Yaskawa INFORM job: A-9-08279-80-90-L.JBI

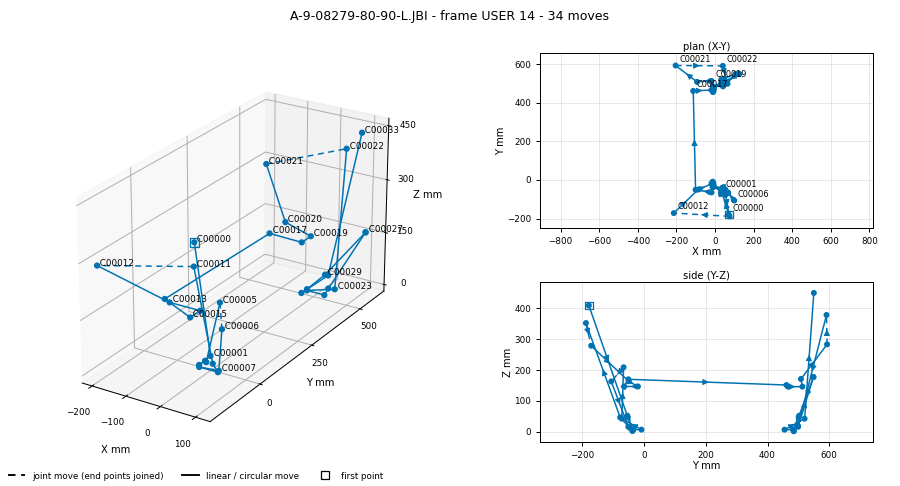
[picture p0: tool path of A-9-08279-80-90-L.JBI in frame USER 14, 34 of 34 moves have a stored position in this frame; points joined in program order, loops and branches not executed]
/JOB
//NAME A-9-08279-80-90-L
///FOLDERNAME PART_420-08279-80
//POS
///NPOS 34,0,34,0,0,0
///USER 14
///TOOL 4
///POSTYPE USER
///RECTAN
///RCONF 1,0,0,0,0,0,0,0,0,0,0,0,0,0,0,0,0,0,0,0,0,0,0,0
C00000=70.970,-178.868,409.213,-165.0000,45.0000,0.0000
C00001=33.224,-54.308,52.156,-165.0000,45.0000,0.0000
C00002=-12.412,-35.347,6.916,178.9966,57.8134,-39.3495
C00003=-12.252,-8.486,6.906,178.9975,57.8083,-39.3460
C00004=32.283,-72.150,42.455,-165.0000,45.0000,0.0000
C00005=68.685,-66.272,209.042,-165.0000,45.0000,0.0000
C00006=99.538,-106.298,163.160,-166.3780,45.3490,-50.4350
C00007=54.868,-50.966,16.241,133.5610,7.6410,-152.0390
C00008=-10.772,-37.614,2.810,126.3860,11.5189,-151.1158
C00009=43.673,-37.455,3.156,126.4274,11.4911,-151.1159
C00010=54.426,-77.432,46.656,126.4293,11.4917,-151.1175
C00011=75.120,-188.373,352.355,175.5546,51.6267,-23.6686
C00012=-213.482,-171.326,278.744,154.4200,34.7310,45.4810
C00013=-87.212,-49.799,163.694,107.6090,9.3560,77.2190
C00014=-17.971,-19.957,146.797,93.4029,5.9535,75.3081
C00015=-18.156,-64.399,146.793,93.4036,5.9529,75.3077
C00016=-100.598,-50.810,170.079,107.6090,9.3560,77.2190
C00017=-112.794,461.129,151.518,107.5190,-7.4490,103.3910
C00018=-17.926,466.306,146.142,97.5705,-4.9534,104.4445
C00019=-17.894,512.947,146.218,97.5696,-4.9493,104.4453
C00020=-92.930,508.215,171.083,107.5190,-7.4490,103.3910
C00021=-203.967,592.873,283.205,107.5190,-7.4490,103.3910
C00022=40.454,590.981,378.479,-169.5230,46.0050,83.6620
C00023=64.926,498.805,18.936,-133.5620,7.6410,152.0390
C00024=-11.073,485.048,2.192,-127.4995,10.8461,151.2305
C00025=41.774,484.768,1.908,-127.7115,11.2204,151.1911
C00026=45.609,498.918,16.234,-144.8388,26.9003,148.6583
C00027=125.350,548.745,177.334,165.0001,45.0004,0.0014
C00028=125.357,548.743,177.335,165.0000,45.0000,0.0000
C00029=33.224,502.241,52.156,165.0000,45.0000,0.0000
C00030=-10.024,483.290,6.806,165.0895,51.2751,6.9885
C00031=-10.615,455.103,6.839,165.1641,51.2621,15.5413
C00032=32.283,520.083,42.455,165.0000,45.0000,0.0000
C00033=107.136,550.049,449.828,165.0032,45.0004,0.0029
///POSTYPE ANGLE
///ANGLE
EC00000=90.0000
EC00001=90.0000
///TOOL 0
EC00002=90.0000
EC00003=90.0000
///TOOL 4
EC00004=90.0000
EC00005=90.0000
EC00006=105.0000
EC00007=105.0000
///TOOL 0
EC00008=105.0000
EC00009=105.0000
EC00010=105.0000
EC00011=105.0000
///TOOL 4
EC00012=135.0000
EC00013=135.0000
///TOOL 0
EC00014=135.0000
EC00015=135.0000
///TOOL 4
EC00016=135.0000
EC00017=135.0000
///TOOL 0
EC00018=135.0000
EC00019=135.0000
///TOOL 4
EC00020=135.0000
EC00021=135.0000
EC00022=105.0000
EC00023=105.0000
///TOOL 0
EC00024=105.0005
EC00025=105.0000
EC00026=105.0000
EC00027=90.0000
///TOOL 4
EC00028=90.0000
EC00029=90.0000
///TOOL 0
EC00030=90.0000
EC00031=90.0000
///TOOL 4
EC00032=90.0000
///TOOL 0
EC00033=90.0000
//INST
///DATE 2021/10/29 11:36
///ATTR SC,RW,RJ
////FRAME USER 14
///GROUP1 RB1
///GROUP2 ST2
NOP
'Path Start: PP1_1
MOVJ C00000 VJ=100.00  +MOVJ EC00000
SMOVL C00001 V=1250.0  +MOVJ EC00001
SMOVL C00002 V=1250.0  +MOVJ EC00002
ARCON ASF#(951)
SMOVL C00003 V=8.5  +MOVJ EC00003
ARCOF AEF#(951)
SMOVL C00004 V=1250.0  +MOVJ EC00004
SMOVL C00005 V=1250.0  +MOVJ EC00005
'Path End
'Path Start: PP48
MOVJ C00006 VJ=100.00  +MOVJ EC00006
SMOVL C00007 V=1250.0  +MOVJ EC00007
SMOVL C00008 V=300.0  +MOVJ EC00008
ARCON ASF#(953)
SMOVL C00009 V=15.7  +MOVJ EC00009
ARCOF AEF#(953)
SMOVL C00010 V=1250.0  +MOVJ EC00010
SMOVL C00011 V=1250.0  +MOVJ EC00011
'Path End
'Path Start: PP47
MOVJ C00012 VJ=100.00  +MOVJ EC00012
SMOVL C00013 V=1250.0  +MOVJ EC00013
SMOVL C00014 V=300.0  +MOVJ EC00014
ARCON ASF#(953)
SMOVL C00015 V=12.7  +MOVJ EC00015
ARCOF AEF#(953)
SMOVL C00016 V=1250.0  +MOVJ EC00016
'Path End
'Path Start: PP42
SMOVL C00017 V=1250.0  +MOVJ EC00017
SMOVL C00018 V=300.0  +MOVJ EC00018
ARCON ASF#(953)
SMOVL C00019 V=12.7  +MOVJ EC00019
ARCOF AEF#(953)
SMOVL C00020 V=1250.0  +MOVJ EC00020
SMOVL C00021 V=1250.0  +MOVJ EC00021
'Path End
'Path Start: PP41
MOVJ C00022 VJ=100.00  +MOVJ EC00022
SMOVL C00023 V=1250.0  +MOVJ EC00023
SMOVL C00024 V=300.0  +MOVJ EC00024
ARCON ASF#(953)
SMOVL C00025 V=15.7  +MOVJ EC00025
ARCOF AEF#(953)
SMOVL C00026 V=1250.0  +MOVJ EC00026
SMOVL C00027 V=1250.0  +MOVJ EC00027
'Path End
'Path Start: PP1
MOVJ C00028 VJ=100.00  +MOVJ EC00028
SMOVL C00029 V=1250.0  +MOVJ EC00029
SMOVL C00030 V=1250.0  +MOVJ EC00030
ARCON ASF#(951)
SMOVL C00031 V=8.5  +MOVJ EC00031
ARCOF AEF#(951)
SMOVL C00032 V=1250.0  +MOVJ EC00032
SMOVL C00033 V=1250.0  +MOVJ EC00033
INC I005
'Path End
END
